{attribute 'qualified_only'}
VAR_GLOBAL
	number:int:=0;
	i: INT:=0;
END_VAR

(* stored: Version 1.1.0.1, ProductVersion 3.1.4024.12
   GVL Random: Id {ccec29ff-c674-42f3-b4cd-daff8107ef2c} *)
